(* CoDeSys 2.3 export: GLOBAL_VARIABLES_MODBUS_MASSAGE.EXP *)

(* Global variable list: Global_Variables_Modbus_Massage *)
VAR_GLOBAL
	T_HMI_Massage AT %MW1.190 :WORD;
	T_BypassMassageStep : WORD;
	T_MassageStep : WORD;
END_VAR
